// TIA Portal V19 export
TYPE "LUC_typeCompleteCommandConfiguration"
// Configure in which states a complete command is possible
// stored: Access Published
   STRUCT
      suspended : Bool := true;   // The Complete control command is taken into account in state Suspended
      execute : Bool := true;   // The Complete control command is taken into account in state Execute
      held : Bool := true;   // The Complete control command is taken into account in state Held
   END_STRUCT;
END_TYPE
